RoboDK station: TM12 Pick and Place.rdk

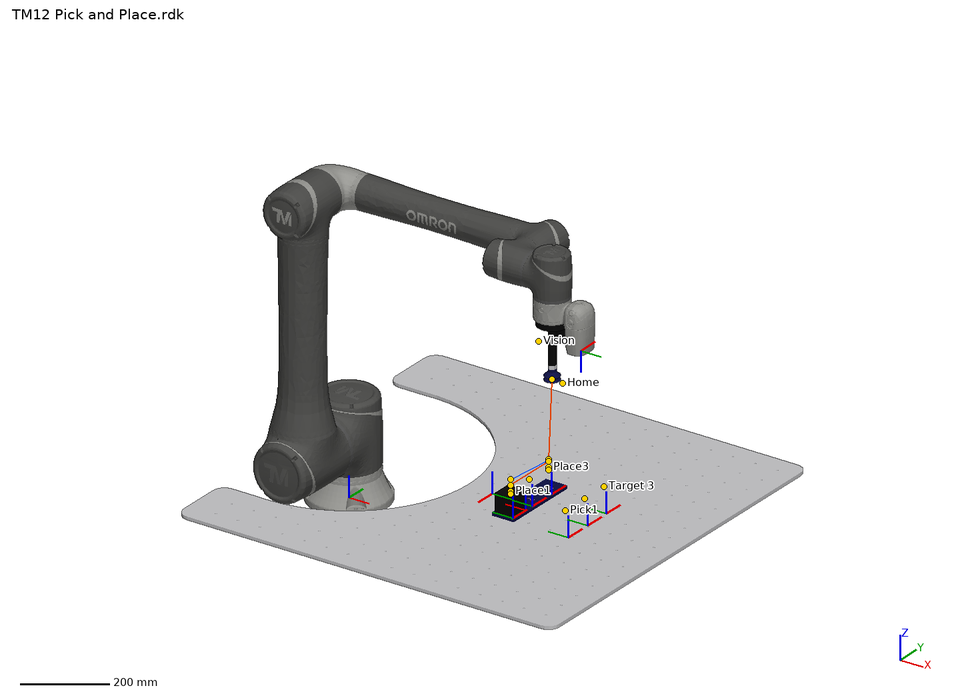
[picture v0: the station drawn from its stored meshes, robots at their saved joint values, targets as dots, program paths as lines]
Station TM12 Station (saved by RoboDK 5.3.5). Poses are relative to the parent item; angles as X-Y-Z fixed-axis rotations.
Station parameters (name, value as stored): IO_1, 1, IO_0, 0
  - frame Omron TM12 Base at (0, 0, -128) mm
    - robot Omron TM12: 6 axes, payload 12 kg, reach 1300 mm, repeatability 0.1 mm, weight 33.3 kg
        modified DH rows (alpha deg, a mm, theta deg, d mm): 0, 0, 0, 165.2; 90, 0, 90, 0; 0, 636.1, 0, 0; 0, 557.9, -90, 156.3; -90, 0, 0, 106; 90, 0, 180, 113.15
        joint limits [-270, -180, -166, -180, -180, -270] to [270, 180, 166, 180, 180, 270]; home [0, 0, 90, -90, 90, 0]; saved at [0, 0, 90, 0, 90, 0]
      - tool TM12 Suction Cup v2, TCP at (0, 0, 146) mm, size 75 x 82.5 x 152 mm, geometry from TM12 Suction Cup v2.step
      - frame Camera Ref at (0, 79, 53) mm
        - camera Camera 1
    - frame Bordet at (392.5, -2.5, 120) mm, rotated rx 0 ry 0 rz -90 deg
      - frame Jig at (50, 127.5, 14) mm, rotated rx 0 ry 0 rz -90 deg
        - object Boks Jig v9 at (0, 0, 0) mm, size 60 x 210 x 9 mm, geometry from Boks Jig v9.step
        - frame Goal 1 at (0, 50, 0) mm, rotated rx 0 ry 0 rz -90 deg
          - target Place1 (Cartesian target) at (25, 25, 50) mm, rotated rx 180 ry 0 rz 0 deg; joints [10.218, -8.622, 137.604, -38.982, 90, 10.218] of Omron TM12
          - target AP (Cartesian target) at (25, 25, 80) mm, rotated rx -180 ry 0 rz 0 deg; joints [10.218, -10.975, 135.54, -34.564, 90, 10.218] of Omron TM12
          - object Box 1 at (0, 0, 0) mm, size 50 x 50 x 50 mm, geometry from Boks 1 v3.step
        - frame Goal 2 at (0, -25, 0) mm, rotated rx 0 ry 0 rz -90 deg
          - target Place2 (Cartesian target) at (25, 25, 50) mm, rotated rx -180 ry 0 rz 0 deg; joints [19.641, -9.288, 138.118, -38.83, 90, 19.641] of Omron TM12
        - frame Goal 3 at (0, -100, 0) mm, rotated rx 0 ry 0 rz -90 deg
          - target Place3 (Cartesian target) at (25, 25, 50) mm, rotated rx 180 ry 0 rz 0 deg; joints [28.543, -8.622, 137.604, -38.982, 90, 28.543] of Omron TM12
          - target AP (Cartesian target) at (25, 25, 70) mm, rotated rx 180 ry 0 rz 0 deg; joints [28.543, -10.228, 136.242, -36.015, 90, 28.543] of Omron TM12
      - frame Box 1 at (100, 277.5, 8) mm, rotated rx 0 ry 0 rz -180 deg
        - target Pick1 (Cartesian target) at (25, 25, 50) mm, rotated rx 180 ry 0 rz 0 deg; joints [7.383, 8.01, 121.9, -39.911, 90, 7.383] of Omron TM12
      - frame Box 2 at (25, 277.5, 8) mm, rotated rx 0 ry 0 rz -180 deg
        - object Box 2 at (0, 0, 0) mm, size 50 x 50 x 50 mm, geometry from Boks 2 v3.step
        - target Target 2 (Cartesian target) at (25, 25, 50) mm, rotated rx 180 ry 0 rz 0 deg; joints [14.192, 7.641, 122.345, -39.985, 90, 14.192] of Omron TM12
      - frame Box 3 at (-50, 277.5, 8) mm, rotated rx 0 ry 0 rz -180 deg
        - object Box 3 at (0, 0, 0) mm, size 50 x 50 x 50 mm, geometry from Boks 3 v3.step
        - target Target 3 (Cartesian target) at (25, 25, 50) mm, rotated rx 180 ry 0 rz 0 deg; joints [20.803, 8.01, 121.9, -39.911, 90, 20.803] of Omron TM12
      - object Omron TM12 Work Surface v1 at (0, 0, 0) mm, size 1000 x 1025 x 8 mm, geometry from Omron TM12 Work Surface v1.step
      - target Home (Cartesian target) at (156.3, 301.4, 422.15) mm, rotated rx 180 ry 0 rz -180 deg; joints [90, -34.737, 125.418, -0.681, 90, 0] of Omron TM12
      - target Vision (Cartesian target) at (0, 127.5, 414) mm, rotated rx 180 ry 0 rz -180 deg; joints [-2.461, -15.13, 102.264, 2.867, 90, 87.539] of Omron TM12
    - target HOME2 (Cartesian target) at (663.9, -156.3, 542.15) mm, rotated rx -180 ry 0 rz 90 deg; joints [0, 0, 90, 0, 90, 0] of Omron TM12
    - target T1 (Cartesian target) at (495, -77.5, 177.5) mm, rotated rx 180 ry 0 rz 90 deg; joints [9.279, -4.887, 135.389, -40.501, 90, 9.279] of Omron TM12
    - target AP1 (Cartesian target) at (495, -77.5, 200) mm, rotated rx 180 ry 0 rz 90 deg; joints [9.279, -6.676, 133.945, -37.268, 90, 9.279] of Omron TM12
    - target T2 (Cartesian target) at (495, 72.5, 177.5) mm, rotated rx 180 ry 0 rz 90 deg; joints [26.538, -4.964, 135.456, -40.491, 90, 26.538] of Omron TM12
    - target AP2 (Cartesian target) at (495, 72.5, 200) mm, rotated rx 180 ry 0 rz 90 deg; joints [26.538, -6.755, 134.01, -37.255, 90, 26.538] of Omron TM12
  - program Home (15 instructions, listed below)
  - program Reset Robot Cell (4 instructions, listed below)
  - program Suction ON (1 instructions, listed below)
  - program Suction OFF (1 instructions, listed below)
  - program Main Porgram (14 instructions, listed below)
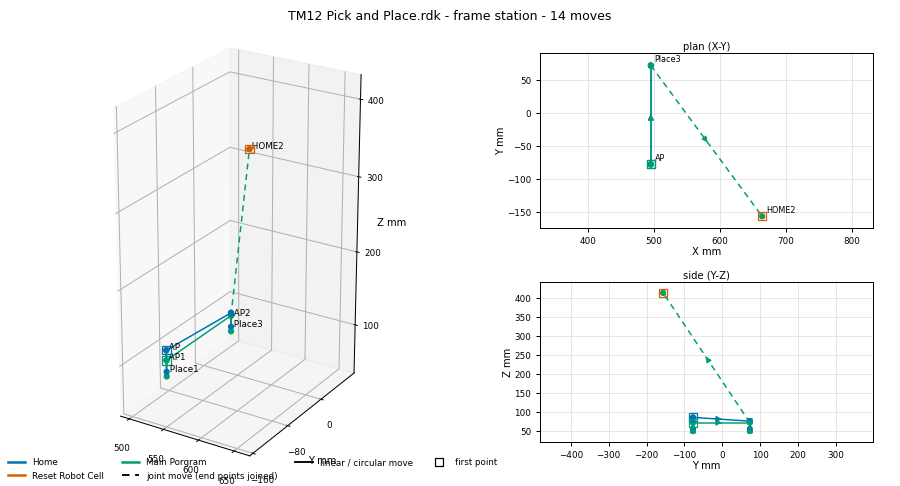
[picture p0: tool path of TM12 Pick and Place.rdk in frame station, 14 of 14 moves have a stored position in this frame; points joined in program order, loops and branches not executed]

--- program Home (robot Omron TM12) ---
  Call Home
  Set Ref.: Goal 1
  Set Tool: TM12 Suction Cup v2
  MoveJ (AP)
  MoveL (Place1)
  Attach to TM12 Suction Cup v2
  Set IO_0=1
  MoveL (AP)
  Set Ref.: Goal 3
  MoveL (AP)
  MoveL (Place3)
  Detach from TM12 Suction Cup v2
  Set IO_0=0
  MoveL (AP)
  Call Reset Robot Cell

--- program Reset Robot Cell (robot Omron TM12) ---
  Set Ref.: Omron TM12 Base
  Set Tool: TM12 Suction Cup v2
  MoveJ (HOME2)
  Replace objects

--- program Suction ON (robot Omron TM12) ---
  Set IO_0=1

--- program Suction OFF (robot Omron TM12) ---
  Set IO_0=0

--- program Main Porgram (robot Omron TM12) ---
  Call Reset Robot Cell
  Set Ref.: Omron TM12 Base
  Set Tool: TM12 Suction Cup v2
  MoveL (AP1)
  MoveJ (T1)
  Attach to TM12 Suction Cup v2
  Call Suction ON
  MoveL (AP1)
  MoveL (Target 19) -> target AP2
  MoveJ (Target 18) -> target T2
  Detach from TM12 Suction Cup v2
  Call Suction OFF
  MoveL (Target 19) -> target AP2
  MoveJ (HOME2)
